FUNCTION_BLOCK FB_LamparaTemporizada_ST
// La lampara se enciende al accionar el pulsador
// La lampara se apaga transcurrido un tiempo encendida
VAR_INPUT
    TiempoEncendido: TIME := T#2S;
    IncrementoTiempo: TIME := T#1S; // Declarado por compatibilidad
END_VAR
VAR_OUTPUT
    TiempoPendiente: TIME;
END_VAR
VAR
    Temporizador: TON;
    Lampara AT %Q*: BOOL;
    Pulsador AT %I*: BOOL;
END_VAR

Temporizador(
    IN := Lampara, 
    PT := TiempoEncendido
    );

IF Pulsador THEN
    Lampara := TRUE;
ELSIF Temporizador.Q THEN
    Lampara := FALSE;
END_IF;

TiempoPendiente := TiempoEncendido - Temporizador.ET;

END_FUNCTION_BLOCK

(* stored: Version 1.1.0.1, ProductVersion 3.1.4024.15
   POU FB_LamparaTemporizada_ST: Id {e4a104bb-8d18-4ef9-8222-84c4e4af6c96}, SpecialFunc None *)
